INTERFACE ITF_LichtSensor

PROPERTY Geblokkeerd : BOOL
GET
END_GET
END_PROPERTY

END_INTERFACE

(* stored: Version 1.1.0.1
   Itf ITF_LichtSensor: Id {9cbb982d-c0cc-4f4d-a4fb-0684eaf937c8}
   Folder Properties: Id {dce72c7d-6ea8-4c05-83c1-b02a44df24d7}
   Property Geblokkeerd: Id {67a4909a-5e1f-453d-9433-d207e28e471d}
   Get Get: Id {0ce39ef6-6409-47d8-b106-7c0f10f9ce35} *)
